// TwinCAT 3 PLC project PLC1
// ProgramVersion: 3.1.4026.24
// libraries:
//   Tc2_MC2, * (Beckhoff Automation GmbH)
//   Tc2_Standard, * (Beckhoff Automation GmbH)
//   Tc2_System, * (Beckhoff Automation GmbH)
//   Tc3_Mc3PlanarMotion, * (Beckhoff Automation GmbH)
//   Tc3_Physics, * (Beckhoff Automation GmbH)
//   Tc3_XPlanarUtility, * (Beckhoff Automation GmbH)
//   XPlanarApplication, * (Beckhoff Automation LLC)
// project tree:
//   GVLs/ GVL.TcGVL (not stored)
//   / PlcTask.TcTTO (not stored)
//   POUs/StationProcesses/ FB_ExtSetpointStation.TcPOU, FB_SimulateProcess.TcPOU
//   POUs/ FB_XPlanarModule.TcPOU, MAIN.TcPOU
//   POUs/Utilities/ ErrorStep.TcPOU (not stored), NextMinorStep.TcPOU (not stored), NextStep.TcPOU
// real-time tasks:
//   TASK XPlanar Task_3: cycle T#250us, priority 1, ADS port 350
//   TASK Job Task: cycle default, priority 2
//   TASK MC-Task (MET): cycle T#2ms, priority 3, ADS port 351
//   TASK MC-Task (MPT): cycle T#10ms, priority 4, ADS port 352
//   TASK PlcTask: cycle T#10ms, priority 20, ADS port 353
// motion (NC):
//   TASK NC-Task 1 SAF: cycle T#2ms, priority 5, ADS port 501
//   TASK NC-Task 1 SVB: cycle T#10ms, priority 9, ADS port 511
//   AXIS VirtualX (id 1)
//     OtherSettings: AllowMotionCmdToSlave=true
//     encoder EncType=1
//     drive DrvType=5
//       Analog: TorqueSetpointScale=10, ScaleFactorActTorque=0.1
//     controller CtrType=1
//       CtrPara: PriorControlFactor=1
//         Observer: BandWidth=20
//   AXIS VirtualY (id 2)
//     OtherSettings: AllowMotionCmdToSlave=true
//     encoder EncType=1
//     drive DrvType=5
//       Analog: TorqueSetpointScale=10, ScaleFactorActTorque=0.1
//     controller CtrType=1
//       CtrPara: PriorControlFactor=1
//         Observer: BandWidth=20
// variable links:
//   PLC1/PLC1 Instance <-> NC-Task 1 SAF/Axes/VirtualX
//     PlcTask Inputs/MAIN.XPlanarTable.ExtSetpointProcess.XAxisNc.NcToPlc <-> Outputs/ToPlc
//     PlcTask Outputs/MAIN.XPlanarTable.ExtSetpointProcess.XAxisNc.PlcToNc <-> Inputs/FromPlc
//   PLC1/PLC1 Instance <-> NC-Task 1 SAF/Axes/VirtualY
//     PlcTask Inputs/MAIN.XPlanarTable.ExtSetpointProcess.YAxisNc.NcToPlc <-> Outputs/ToPlc
//     PlcTask Outputs/MAIN.XPlanarTable.ExtSetpointProcess.YAxisNc.PlcToNc <-> Inputs/FromPlc
//   PLC1/PLC1 Instance <-> XPlanar MC Project/Axes/Mover4220_1
//     PlcTask Inputs/MAIN.XPlanarTable.Movers[1]._Mover.MCTOPLC/ACT <-> McToPlc/ACT
//     PlcTask Inputs/MAIN.XPlanarTable.Movers[1]._Mover.MCTOPLC/COORDMODE <-> McToPlc/COORDMODE
//     PlcTask Inputs/MAIN.XPlanarTable.Movers[1]._Mover.MCTOPLC/SET <-> McToPlc/SET
//     PlcTask Inputs/MAIN.XPlanarTable.Movers[1]._Mover.MCTOPLC/SETONTRACK <-> McToPlc/SETONTRACK
//     PlcTask Inputs/MAIN.XPlanarTable.Movers[1]._Mover.MCTOPLC/STD <-> McToPlc/STD
//     PlcTask Outputs/MAIN.XPlanarTable.Movers[1]._Mover.PLCTOMC/STD <-> PlcToMc/STD
//   PLC1/PLC1 Instance <-> XPlanar MC Project/Axes/Mover4220_2
//     PlcTask Inputs/MAIN.XPlanarTable.Movers[2]._Mover.MCTOPLC/ACT <-> McToPlc/ACT
//     PlcTask Inputs/MAIN.XPlanarTable.Movers[2]._Mover.MCTOPLC/COORDMODE <-> McToPlc/COORDMODE
//     PlcTask Inputs/MAIN.XPlanarTable.Movers[2]._Mover.MCTOPLC/SET <-> McToPlc/SET
//     PlcTask Inputs/MAIN.XPlanarTable.Movers[2]._Mover.MCTOPLC/SETONTRACK <-> McToPlc/SETONTRACK
//     PlcTask Inputs/MAIN.XPlanarTable.Movers[2]._Mover.MCTOPLC/STD <-> McToPlc/STD
//     PlcTask Outputs/MAIN.XPlanarTable.Movers[2]._Mover.PLCTOMC/STD <-> PlcToMc/STD
//   PLC1/PLC1 Instance <-> XPlanar MC Project/Groups/Environment
//     PlcTask Inputs/XPlanar.Environment.MCTOPLC_STD <-> McToPlc/STD
//   PLC1/PLC1 Instance <-> XPlanar MC Project/Groups/Track1
//     PlcTask Inputs/MAIN.XPlanarTable.Tracks[1]._Track.MCTOPLC_STD <-> McToPlc/STD
//   PLC1/PLC1 Instance <-> XPlanar MC Project/Groups/Track2
//     PlcTask Inputs/MAIN.XPlanarTable.Tracks[2]._Track.MCTOPLC_STD <-> McToPlc/STD
//   PLC1/PLC1 Instance <-> XPlanar MC Project/Groups/XPlanar
//     PlcTask Inputs/XPlanar.Group.MCTOPLC_STD <-> McToPlc/STD
//   TcCOM Objects/XPlanar/Mover4220_1 <-> XPlanar MC Project/Axes/Mover4220_1
//     InputsFromNC3/NC3ToHW <-> McToIo/STD
//     OutputsToNC3/HWToNC3 <-> IoToMc/STD
//   TcCOM Objects/XPlanar/Mover4220_2 <-> XPlanar MC Project/Axes/Mover4220_2
//     InputsFromNC3/NC3ToHW <-> McToIo/STD
//     OutputsToNC3/HWToNC3 <-> IoToMc/STD

// ---- POUs/StationProcesses/FB_ExtSetpointStation.TcPOU
FUNCTION_BLOCK FB_ExtSetpointStation IMPLEMENTS I_StationProcess
VAR
	//NC PTP Axis Vars
	XAxisNc 		: AXIS_REF;
	YAxisNc 		: AXIS_REF;
	EnableXAxis 	: MC_Power;
	EnableYAxis 	: MC_Power;
	MoveXAxis		: MC_MoveAbsolute;
	MoveYAxis		: MC_MoveAbsolute;
	
	XAxisVelo		: LREAL := 250;
	YAxisVelo		: LREAL := 250;
	XAxisPos		: LREAL;
	YAxisPos		: LREAL;
	XAxisMove		: BOOL;
	YAxisMove		: BOOL;
	
	//Internal Vars
	ProcessState 	: DINT;
	movervector	 	: movervector;
	initsequence	: DINT;
END_VAR

METHOD Execute : BOOL
VAR_INPUT
	Mover	: XPlanarApplication.I_XPlanarMover;
END_VAR

VAR_INST
	CommandResult 	: I_PlanarTaskResult;
	MoverVectorPos 	: MoverVector;
	MoverVectorVel 	: MoverVector;
	MoverVectorAcc	: MoverVector;
	RunExtSp		: BOOL;
END_VAR

CASE ProcessState OF
	0: //Init
		//Could verify XAxis and YAxis are are valid starting positions here***
		ProcessState := 10;

	10: //Move to Target Position
		XAxisPos  := 50;
		YAxisPos  := 50;
		XAxisMove := TRUE;
		YAxisMove := TRUE;
		RunExtSp  := TRUE;
		IF MoveXAxis.Busy AND MoveYAxis.Busy THEN
			XAxisMove	 := FALSE;
			YAxisMove	 := FALSE;
			ProcessState := 20;
		END_IF

	20: //Wait for NC move to complete
		IF MoveXAxis.Done AND MoveYAxis.Done THEN
			ProcessState := 30;
		END_IF

	30: //Return to Start Pos
		XAxisPos  := 0;
		YAxisPos  := 0;
		XAxisMove := TRUE;
		YAxisMove := TRUE;
		RunExtSp  := TRUE;
		IF MoveXAxis.Busy AND MoveYAxis.Busy THEN
			XAxisMove	 := FALSE;
			YAxisMove	 := FALSE;
			ProcessState := 40;
		END_IF

	40: //Wait for NC move to complete
		IF MoveXAxis.Done AND MoveYAxis.Done THEN
			ProcessState := 50;
		END_IF

	50:
		IF MoverVectorPos.x = 0 AND MoverVectorPos.y = 0 AND MoverVectorVel.x = 0 AND MoverVectorVel.y = 0 THEN
			RunExtSp := FALSE;

			//Take mover out of external setpoint mode
			CommandResult := Mover.MoveCommand.StopExternalSp();
			// program has finished
			IF CommandResult.Done THEN
				Execute := TRUE;
				ProcessState := 0;
			END_IF
		END_IF
END_CASE

IF RunExtSp THEN
	MoverVectorPos.x := XAxisNc.NcToPlc.SetPos;
	MoverVectorPos.y := YAxisNc.NcToPlc.SetPos;
	MoverVectorVel.x := XAxisNc.NcToPlc.SetVelo;
	MoverVectorVel.y := YAxisNc.NcToPlc.SetVelo;
	MoverVectorAcc.x := XAxisNc.NcToPlc.SetAcc;
	MoverVectorAcc.y := YAxisNc.NcToPlc.SetAcc;
	CommandResult	 := Mover.MoveCommand.RunExternalSpRelativeMode(MoverVectorPos, MoverVectorVel, MoverVectorAcc);
END_IF

//X Axis NC Move
MoveXAxis(Axis		   := XAxisNc,
		  Execute	   := XAxisMove,
		  Position	   := XAxisPos,
		  Velocity	   := XAxisVelo,
		  Acceleration := XAxisVelo * 10,
		  Deceleration := XAxisVelo * 10,
		  Jerk		   := XAxisVelo * 100,
		  BufferMode   := MC_BufferMode.MC_Aborting);

//Y Axis NC Move
MoveYAxis(Axis		   := YAxisNc,
		  Execute	   := YAxisMove,
		  Position	   := YAxisPos,
		  Velocity	   := YAxisVelo,
		  Acceleration := YAxisVelo * 10,
		  Deceleration := YAxisVelo * 10,
		  Jerk		   := YAxisVelo * 100,
		  BufferMode   := MC_BufferMode.MC_Aborting);
END_METHOD

(* Basic component initialization logic*)
METHOD Initialize : BOOL

VAR
	
END_VAR
CASE initsequence OF
	0:
		EnableXAxis(
			Axis := XAxisNc,
			Enable := TRUE,
			Enable_Positive:= TRUE,
			Enable_Negative:= TRUE,
			Override := 100.0);
		
		EnableYAxis(
			Axis := YAxisNc,
			Enable := TRUE,
			Enable_Positive:= TRUE,
			Enable_Negative:= TRUE,
			Override := 100.0);
			
		IF EnableXAxis.Status AND EnableYAxis.Status THEN
			initsequence := 10;
		END_IF
		
	10:
	Initialize := TRUE;
	
END_CASE
END_METHOD

END_FUNCTION_BLOCK

// ---- POUs/FB_XPlanarModule.TcPOU
FUNCTION_BLOCK FB_XPlanarModule
VAR CONSTANT
	MoverCount	 : UDINT := 2;
	TrackCount	 : UDINT := 2;
	StationCount : UDINT := 2;
END_VAR

VAR
	XPlanarSystem	   : FB_Component_XPlanar;
	Movers			   : ARRAY[1..MoverCount] OF FB_XPlanarMover;
	Tracks			   : ARRAY[1..TrackCount] OF FB_XPlanarTrackSegment;
	Stations		   : ARRAY[1..StationCount] OF FB_XPlanarStationBase;
	ExtSetpointProcess : FB_ExtSetpointStation;
	SimulateProcess	   : FB_SimulateProcess := (ProcessTime := 1.5);
	InitState		   : (CheckForXPlanarInit, UpdateDynamics, SetStationParameters, Initialized);
END_VAR

METHOD CyclicLogic : BOOL
VAR
	i : UDINT;
END_VAR
VAR_INST
	MoverGapCheck: LREAL;
	GlobalGapUpdate: BOOL;
	testers	: UDINT;
	TestMove	: BOOL;
	TaskResult	: I_PlanarTaskResult;
END_VAR
XPlanarSystem.CyclicLogic();
IF NOT XPlanarSystem.Initialized THEN
	RETURN;
END_IF

//Add any logic that needs to be called every cycle here
END_METHOD

METHOD Disable : BOOL
VAR_INST
	CommandResult	: I_PlanarTaskResult;
END_VAR
CommandResult := XPlanarSystem.Abort(); // Stop Motion and Disable All Movers
IF CommandResult.Done THEN
	Disable := TRUE;
END_IF
END_METHOD

METHOD Execute : BOOL
VAR
	i : UDINT;
END_VAR
//The XPlanar system is now 'running' put necessary run logic here

FOR i := 1 TO XPlanar.StationCount DO
	Stations[i].Execute();
END_FOR
END_METHOD

METHOD Initialize : BOOL
VAR_INST
	i			: UDINT;
END_VAR
CASE InitState OF
	CheckForXPlanarInit: // Init Vars
		Initialize := FALSE;
		
		//Make sure the XPlanar motion system has initialized
		IF XPlanarSystem.Initialized THEN
			InitState := UpdateDynamics;
		END_IF

	UpdateDynamics: // Assign Initial Application Mover Dynamics
		FOR i := 1 TO XPlanar.MoverCount DO
			ip.Movers[i].Gap						:= 200;
			ip.Movers[i].Dynamics.Movement.Velocity := GVL.MoverVelo;
			ip.Movers[i].Dynamics.Movement.Accel	:= GVL.MoverVelo * 10;
			ip.Movers[i].Dynamics.Movement.Decel	:= GVL.MoverVelo * 10;
			ip.Movers[i].Dynamics.Movement.Jerk		:= GVL.MoverVelo * 100;
			ip.Movers[i].Dynamics.Rotation.Velocity := GVL.MoverSpinVelo;
			ip.Movers[i].Dynamics.Rotation.Accel	:= GVL.MoverSpinVelo * 10;
			ip.Movers[i].Dynamics.Rotation.Decel	:= GVL.MoverSpinVelo * 10;
			ip.Movers[i].Dynamics.Rotation.Jerk		:= GVL.MoverSpinVelo * 100;
		END_FOR

		InitState := SetStationParameters;

	SetStationParameters:
		IF SetupStations() THEN
			InitState := Initialized;
		END_IF
		
		//Initialize station processes if necessary
		ExtSetpointProcess.Initialize();

	Initialized: // Init Complete
		Initialize := TRUE;
END_CASE
END_METHOD

METHOD Recovery : BOOL
VAR_INST
	RecoverState	: UDINT;
	ipResult		: ARRAY[1..MoverCount] OF I_PlanarTaskResult;
	ErrorMoverId, i : UDINT;
	ItemsOk			: BOOL;
END_VAR
CASE RecoverState OF
	0: // Init Vars
		Recovery := FALSE;
		i := 1;
		NextStep(RecoverState);
		
	10: // All Movers Join Closest Track
		IF i <= XPlanar.MoverCount THEN
			ipResult[i] := Movers[i].MoveCommand.JoinClosestTrack(FALSE);
			IF ipResult[i].Done THEN
				NextMinorStep(RecoverState);
			ELSIF ipResult[i].Error THEN
				ErrorStep(RecoverState);
			END_IF
		ELSE
			i := 1;
			NextStep(RecoverState);
		END_IF

	11: //Check Mover Count
		IF i <= XPlanar.MoverCount THEN
			i	   := i + 1;
			RecoverState := 10;
		ELSE
			i := 1;
			NextStep(RecoverState);
		END_IF

	20: // Sort and send Movers to Stations
		FOR i := 1 TO XPlanar.MoverCount DO
			ipResult[i] := Movers[i].MoveCommand.SendToStation(Stations[1]);
		END_FOR

		NextStep(RecoverState);

	30: // Wait For Mover to Move
		ItemsOk := TRUE;
		FOR i := 1 TO XPlanar.MoverCount DO
			IF NOT ipResult[i].Busy THEN
				ItemsOk := FALSE;
			END_IF

			IF ipResult[i].Error THEN
				ErrorMoverId := i;
				ErrorStep(RecoverState);
			END_IF
		END_FOR

		IF ItemsOk THEN
			ErrorMoverId := 0;
			NextStep(RecoverState);
		END_IF

	40: // Complete
		RecoverState		 := 0;
		ErrorMoverId := 0;
		Recovery	 := TRUE;
END_CASE
END_METHOD

METHOD Reset : BOOL
VAR_INST
	ResettingState : UDINT;
	i			   : UDINT;
	ResetOk		   : BOOL;
	ResetError	   : BOOL;
	CommandResult  : I_PlanarTaskResult;
END_VAR
CASE ResettingState OF
	0: // Init Vars
		Reset := FALSE;
		NextStep(ResettingState);

	10: // Reset Table 
		IF XPlanarSystem.Reset().Done THEN
			NextStep(ResettingState);
		END_IF

	20: // Reset Stations
		FOR i := 1 TO StationCount DO
			ip.Stations[i].Reset();
		END_FOR

		NextStep(ResettingState);

	30: // Enable Movers
		CommandResult := XPlanarSystem.EnableMovers();
		IF CommandResult.Done THEN
			NextStep(ResettingState);
		ELSIF CommandResult.Error THEN
			ErrorStep(ResettingState);
		END_IF

	40: // Add Movers To Group
		CommandResult := XPlanarSystem.AddMoversToGroup();
		IF CommandResult.Done THEN
			NextStep(ResettingState);
		ELSIF CommandResult.Error THEN
			ErrorStep(ResettingState);
		END_IF

	50: // Enable Tracks
		CommandResult := XPlanarSystem.EnableTracks();
		IF CommandResult.Done THEN
			NextStep(ResettingState);
		ELSIF CommandResult.Error THEN
			ErrorStep(ResettingState);
		END_IF

	60: // Add Tracks To Group
		CommandResult := XPlanarSystem.AddTracksToGroup();
		IF CommandResult.Done THEN
			NextStep(ResettingState);
		ELSIF CommandResult.Error THEN
			ErrorStep(ResettingState);
		END_IF

	70: // Enable Group
		CommandResult := XPlanarSystem.EnableGroup();
		IF CommandResult.Done THEN
			NextStep(ResettingState);
		ELSIF CommandResult.Error THEN
			ErrorStep(ResettingState);
		END_IF

	80: // Complete
		Reset  := TRUE;
		ResettingState := 0;
END_CASE
END_METHOD

METHOD PRIVATE SetupStations : BOOL
// Setup Station 1
Stations[1].ID := 1;
Stations[1].TrackID := 1;
Stations[1].Position.SetValuesXYC(120, 60, 0);
Stations[1].NextStation := Stations[2];
Stations[1].Process := SimulateProcess; //Assign a custom process to the station



// Setup Station 2
Stations[2].ID := 2;
Stations[2].TrackID := 2;
Stations[2].Position.SetValuesXYC(120, 360, 0);
Stations[2].NextStation := Stations[1];
Stations[2].Process := ExtSetpointProcess; //Assign a custom process to the station


SetupStations:=TRUE;
END_METHOD

END_FUNCTION_BLOCK

// ---- POUs/StationProcesses/FB_SimulateProcess.TcPOU
FUNCTION_BLOCK FB_SimulateProcess IMPLEMENTS I_StationProcess
VAR
	_ProcessTime	: TIME;
END_VAR

METHOD Execute : BOOL
VAR_INPUT
	Mover	: XPlanarApplication.I_XPlanarMover;
END_VAR

VAR_INST
	SimulateTimer: TON;
END_VAR
SimulateTimer(IN := Mover <> 0, PT := _ProcessTime);
IF SimulateTimer.Q THEN
	SimulateTimer(IN := FALSE);
	Execute := TRUE; //Set Execute to TRUE when process is complete and station base will send mover to next station.
END_IF
END_METHOD

PROPERTY ProcessTime : LREAL
SET
_ProcessTime := TO_TIME(ProcessTime * 1000);
END_SET
END_PROPERTY

END_FUNCTION_BLOCK

// ---- POUs/Utilities/NextStep.TcPOU
FUNCTION NextStep : UDINT
VAR_IN_OUT
	StateVar : UDINT;
END_VAR

NextStep := StateVar := ((StateVar / 10) * 10) + 10;

END_FUNCTION

// ---- POUs/MAIN.TcPOU
PROGRAM MAIN
VAR
	XPlanarTable  : FB_XPlanarModule;
	Initialize	  : BOOL;
	Reset		  : BOOL; // Reset and Execute System
	Start		  : BOOL; // Run the system
	Halt		  : BOOL; // Avoid Disabling while spinning, otherwise physical sqauring of mover is required
	MachineState  : (Startup,
		InitSystem,
		ResetSystem,
		Recover,
		Ready,
		Run,
		Disable);
	trig  : R_TRIG;
	count: INT;
END_VAR

//This project is a bacis example that shows how to use the External Setpoint function of a mover 
//in relative mode as a way to add some custom movement without leaving the track network
//It is a working sample where the process attached to station 2 commands the mover away from the track and back before continuing to the next station
//The External Setpoint logic is the Execute method of FB_ExtSetpointStation


//Keep all XPlanar motion system objects up to date every cycle
XPlanarTable.CyclicLogic();


// "Machine" Sequence
CASE MachineState OF
	Startup:	
		IF Initialize THEN
			Initialize := FALSE;
			MachineState := InitSystem;
		END_IF
	
	InitSystem:	
		IF XPlanarTable.Initialize() THEN
			MachineState := ResetSystem;
		END_IF
	
	ResetSystem:	
		IF Reset AND_THEN XPlanarTable.Reset() THEN
			Reset := FALSE;
			MachineState := Recover;
		END_IF
	
	Recover:	
		IF XPlanarTable.Recovery() THEN
			MachineState := Ready;
		END_IF
		
	Ready:
		IF Start THEN
			MachineState := Run;
		END_IF
	
	Run: 
		XPlanarTable.Execute();
	
	Disable:	
		IF XPlanarTable.Disable() THEN
			MachineState := 0;
		END_IF
END_CASE

IF Halt OR trig.Q THEN
	MachineState := Disable;
	Halt := FALSE;
END_IF

END_PROGRAM
